// Generic interface that defines the basic properties and methods of an object in the FisoThemes Standard Library.
INTERFACE FsI_Object EXTENDS FsI_Unknown

// Pointer to the object in memory.
PROPERTY Address : FsT_Ptr
GET
END_GET
END_PROPERTY

// Represents the path to the object.
PROPERTY InstancePath : FsT_LStr
GET
END_GET
END_PROPERTY

// Checks if the current object is the same as (reference-wise) object as the input object.
METHOD Is : BOOL
VAR_INPUT
	ipObject : FsI_Object;
END_VAR
END_METHOD

// Memory area that the object is allocated in.
PROPERTY MemoryArea : FsT_MemArea
GET
END_GET
END_PROPERTY

//  Size of the object in bytes.
PROPERTY Size : FsT_Size
GET
END_GET
END_PROPERTY

// Converts this object to a string representation.
METHOD ToString : FsT_LStr
END_METHOD

// A string that represents the type of the object.
PROPERTY TypeName : FsT_Str
GET
END_GET
END_PROPERTY

END_INTERFACE

(* stored: Version 1.1.0.1, ProductVersion 3.1.4024.4
   Itf FsI_Object: Id {201a7385-47ee-481f-a692-da4578c9197f}
   Folder Methods: Id {603824c2-a15f-4b68-9f03-78f8bd8cf16c}
   Folder Properties: Id {6528398b-04f5-484f-a69c-a3efa596900f}
   Property Address: Id {4ac6af2f-263b-4789-aa5c-4534d7e3601d}
   Get Get: Id {fb480715-7e3a-4ba1-b3a2-ce287c463598}
   Property InstancePath: Id {ad2ab2a4-30f3-4204-901b-e2de4905e992}
   Get Get: Id {ee4fdb97-c081-484e-a6ea-b8e30569360a}
   Method Is: Id {78d3b0be-7a2f-4ba2-950a-f12e5b6bcb3f}
   Property MemoryArea: Id {547eaac8-abd9-4938-856a-d7d56950eb21}
   Get Get: Id {091cd4dc-96c4-45e4-bcf6-ba1f8a1218fb}
   Property Size: Id {65368e23-d7cc-4f00-9614-fa13d1015bcf}
   Get Get: Id {745bf69d-9e54-4f66-92c5-6afce78353b6}
   Method ToString: Id {dc567948-de95-41dc-a569-aaa1494a51b5}
   Property TypeName: Id {ffb197d2-6d6a-47ea-889c-6981af5783f6}
   Get Get: Id {3fd8aecb-d27d-41c3-885f-c5c5209402fa} *)
